Omron CX-Programmer project NewProject (CX-Programmer 9.73)

# PLC TUBES_1: CP1H XA

## Global symbols (name address type ; comment)
0.00 BOOL  ; PB_ON
0.01 BOOL  ; PB_OFF
100.00 BOOL  ; Lampu Hijau Simpang 1
100.01 BOOL  ; Lampu Kuning Simpang 1
100.02 BOOL  ; Lampu Merah Simpang 1
100.03 BOOL  ; Lampu Hijau Simpang 2
100.04 BOOL  ; Lampu Kuning Simpang 2
100.05 BOOL  ; Lampu Merah Simpang 2
100.06 BOOL  ; Lampu Hijau Simpang 3
100.07 BOOL  ; Lampu Kuning Simpang 3
100.08 BOOL  ; Lampu Merah Simpang 3
100.09 BOOL  ; Lampu Hijau Simpang 4
100.10 BOOL  ; Lampu Kuning Simpang 4
100.11 BOOL  ; Lampu Merah Simpang 4
101.00 BOOL  ; Lampu Kuning Simpang 3
101.01 BOOL  ; Lampu Merah Simpang 3
101.02 BOOL  ; Lampu Hijau Simpang 4
101.03 BOOL  ; Lampu Kuning Simpang 4
101.04 BOOL  ; Lampu Merah Simpang 4
10.00 BOOL  ; System ON
10.01 BOOL  ; RTC 0N
A351 CHANNEL  ; HOUR
A354 CHANNEL  ; DAY
W0.00 BOOL  ; Running

## Program NewProgram1 (cyclic task 0)

### Section Section1

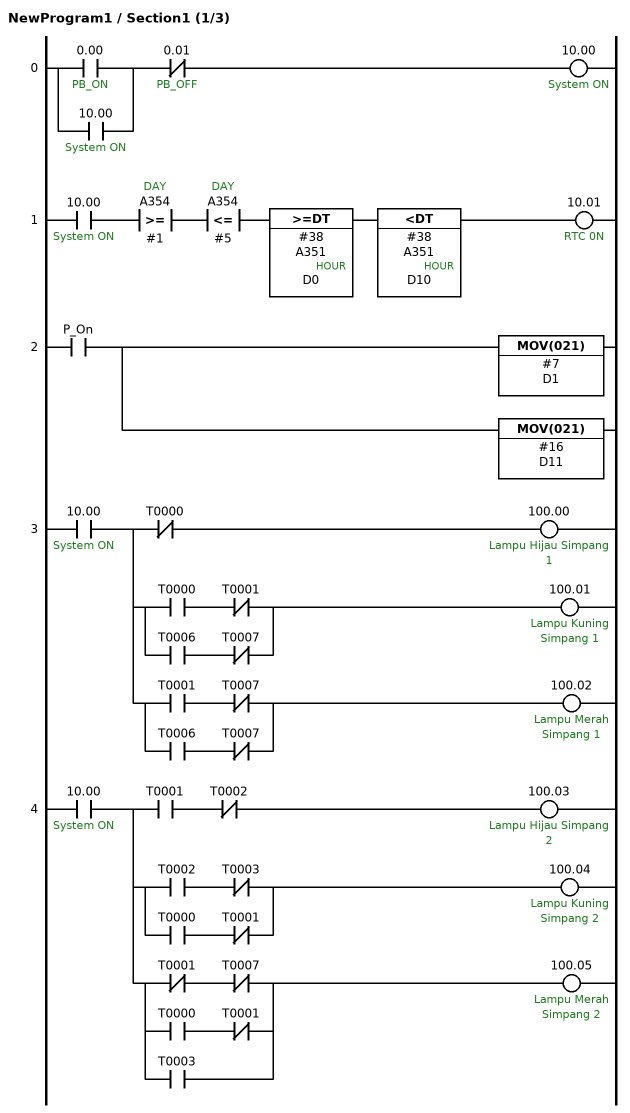
; rung 0
LD 0.00  ; PB_ON
OR 10.00  ; System ON
ANDNOT 0.01  ; PB_OFF
OUT 10.00  ; System ON
; rung 1
LD 10.00  ; System ON
AND>=(325) A354 #1  ; DAY
AND<=(315) A354 #5  ; DAY
AND>=DT(346) #38 A351 D0  ; HOUR
AND<DT(343) #38 A351 D10  ; HOUR
OUT 10.01  ; RTC 0N
; rung 2
LD P_On
MOV(021) #7 D1
MOV(021) #16 D11
; rung 3
LD 10.00  ; System ON
OUT TR0
ANDNOT T0000
OUT 100.00  ; Lampu Hijau Simpang 1
LD TR0
LD T0000
ANDNOT T0001
LD T0006
ANDNOT T0007
ORLD
ANDLD
OUT 100.01  ; Lampu Kuning Simpang 1
LD TR0
LD T0001
ANDNOT T0007
LD T0006
ANDNOT T0007
ORLD
ANDLD
OUT 100.02  ; Lampu Merah Simpang 1
; rung 4
LD 10.00  ; System ON
OUT TR0
AND T0001
ANDNOT T0002
OUT 100.03  ; Lampu Hijau Simpang 2
LD TR0
LD T0002
ANDNOT T0003
LD T0000
ANDNOT T0001
ORLD
ANDLD
OUT 100.04  ; Lampu Kuning Simpang 2
LD TR0
LDNOT T0001
ANDNOT T0007
LD T0000
ANDNOT T0001
ORLD
OR T0003
ANDLD
OUT 100.05  ; Lampu Merah Simpang 2

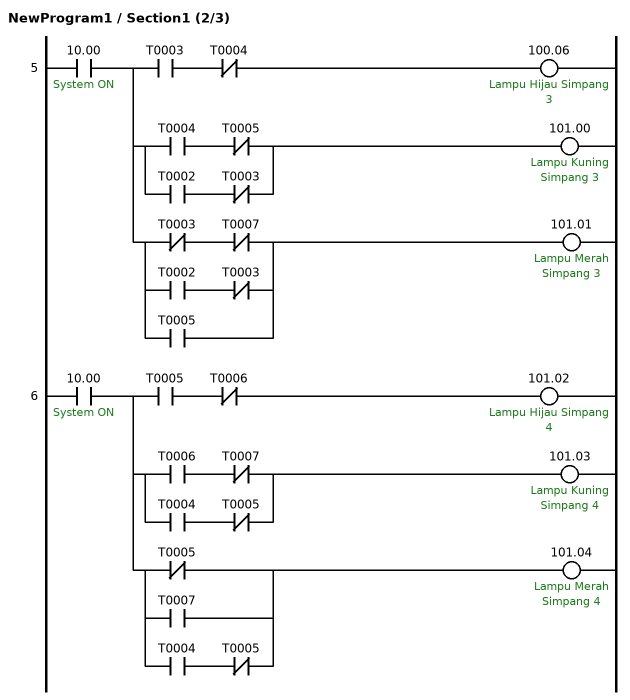
; rung 5
LD 10.00  ; System ON
OUT TR0
AND T0003
ANDNOT T0004
OUT 100.06  ; Lampu Hijau Simpang 3
LD TR0
LD T0004
ANDNOT T0005
LD T0002
ANDNOT T0003
ORLD
ANDLD
OUT 101.00  ; Lampu Kuning Simpang 3
LD TR0
LDNOT T0003
ANDNOT T0007
LD T0002
ANDNOT T0003
ORLD
OR T0005
ANDLD
OUT 101.01  ; Lampu Merah Simpang 3
; rung 6
LD 10.00  ; System ON
OUT TR0
AND T0005
ANDNOT T0006
OUT 101.02  ; Lampu Hijau Simpang 4
LD TR0
LD T0006
ANDNOT T0007
LD T0004
ANDNOT T0005
ORLD
ANDLD
OUT 101.03  ; Lampu Kuning Simpang 4
LD TR0
LDNOT T0005
OR T0007
LD T0004
ANDNOT T0005
ORLD
ANDLD
OUT 101.04  ; Lampu Merah Simpang 4

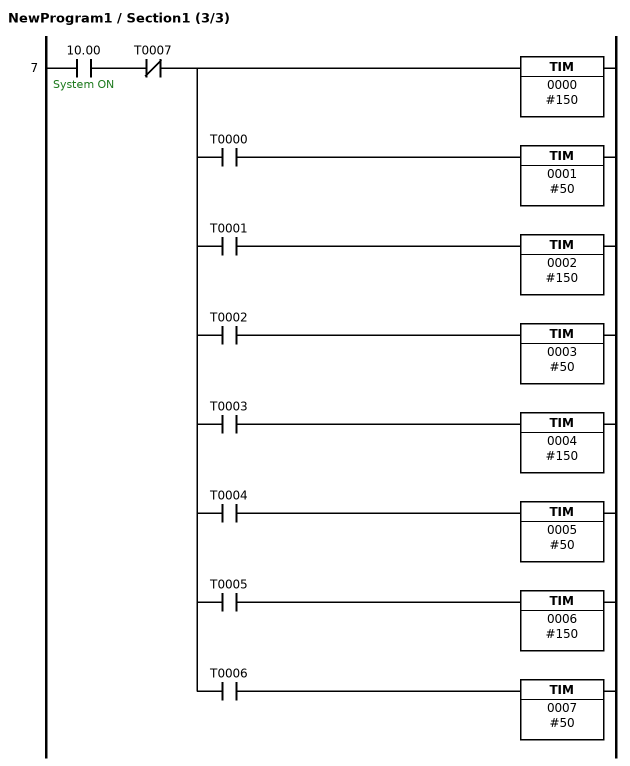
; rung 7
LD 10.00  ; System ON
ANDNOT T0007
OUT TR0
TIM 0000 #150
AND T0000
TIM 0001 #50
LD TR0
AND T0001
TIM 0002 #150
LD TR0
AND T0002
TIM 0003 #50
LD TR0
AND T0003
TIM 0004 #150
LD TR0
AND T0004
TIM 0005 #50
LD TR0
AND T0005
TIM 0006 #150
LD TR0
AND T0006
TIM 0007 #50

### Section END
; rung 0
END(001)